(* IEC 61131-3 sources: codescribe/GraphicalTesting/SafetyPLC/application, 2 files *)

(* ---- EVL.gvl.st ---- *)
(* THIS EVL IS AUTOGENERATED. DO NOT MODIFY THESE ATTRIBUTES. *)
{attribute 'location' := '16#800' }
{attribute 'linkalways'}
{attribute 'qualified_only'}
VAR_GLOBAL

END_VAR

(* ---- PLC_PRG.st ---- *)
PROGRAM PLC_PRG
VAR

END_VAR

// --- BEGIN IMPLEMENTATION ---
